Fanuc KAREL source: mth_sqrt.kl

PROGRAM mth_sqrt
%NOBUSYLAMP
%NOLOCKGROUP

VAR
	out_reg : INTEGER
	val : REAL
%from tpe.klh %import get_int_arg,get_real_arg
%from registers.klh %import set_real
%from math.builtins.klh %import sqrt

BEGIN
	val = tpe__get_real_arg(1)
	out_reg = tpe__get_int_arg(2)
	registers__set_real(out_reg, math__sqrt(val))
END mth_sqrt
